FUNCTION_BLOCK FB_PLCopenCall_Test EXTENDS FB_TestSuite
VAR_INPUT
END_VAR
VAR_OUTPUT
END_VAR
VAR
END_VAR

// Copyright (c) 2024 Loupe (https://loupe.team), provided under the MIT License.

Call();
Clear();
Exec();
Start();

METHOD Call
VAR
    call : PLCopenCall;
    command : PLCopenCommand;
END_VAR
// Copyright (c) 2024 Loupe (https://loupe.team), provided under the MIT License.

(*STweep.Disable*)

TEST('PLCopenCallIdle');


	AssertFalse(Condition := call.Busy, Message := 'Busy should be false as default');
	AssertFalse(Condition := call.Done, Message := 'Done should be false as default');
	AssertFalse(Condition := call.Error, Message := 'Error should be false as default');
	
	call.Exec(command);
	AssertTrue(Condition := call.Busy, Message := 'Busy should be true after first exec');
	AssertFalse(Condition := call.Done, Message := 'Done should be false after first exec');
	AssertFalse(Condition := call.Error, Message := 'Error should be false as default');
	AssertEquals_DINT(Expected := PLCopenStatusBase.BUSY, Actual := call.Status, Message := 'Status should be FUB Working');

// new command

// this command aborted

// cleanup

// done

// working

// aborted

// TODO multiple calls
TEST_FINISHED();
END_METHOD

METHOD Clear
VAR
    call : PLCopenCall();
    status : PLCopenStatusBase;
END_VAR
// Copyright (c) 2024 Loupe (https://loupe.team), provided under the MIT License.

(*STweep.Disable*)

TEST('Clear');
	call.Execute := TRUE;
	call();
	status := call.Clear();
	AssertFalse(call.Execute, Message := 'Execute should not be true');
	AssertEquals_INT(Expected := PLCopenStatusBase.NOT_ENABLED, Actual := status, Message := 'Call status should be not enabled');
TEST_FINISHED();
END_METHOD

METHOD Errored
VAR_INPUT
END_VAR
// Copyright (c) 2024 Loupe (https://loupe.team), provided under the MIT License.

(*STweep.Disable*)
END_METHOD

METHOD Exec
VAR
    call : PLCopenCall();
    command1 : PLCopenCommand();
    command2 : PLCopenCommand();
END_VAR
// Copyright (c) 2024 Loupe (https://loupe.team), provided under the MIT License.

(*STweep.Disable*)

TEST('Exec');
	call.Exec(command1);
	AssertTrue(call.Execute, Message := 'Execute should be true');
	
	call.Exec(command2);
	AssertTrue(call.Execute, Message := 'Execute should still be true, second command should abort first');
	AssertFalse(command1.Execute, Message := 'Execute should not be true on first command');
TEST_FINISHED();
END_METHOD

METHOD Start
VAR
    call : PLCopenCall();
    command1 : PLCopenCommand();
    command2 : PLCopenCommand();
END_VAR
// Copyright (c) 2024 Loupe (https://loupe.team), provided under the MIT License.

(*STweep.Disable*)

TEST('Start');
    // TODO check cancelling previous command
	
	// NOTE: since Start is just a wrapper around Exec, these tests are the same as Exec
	call.Start(command1);
	AssertTrue(call.Execute, Message := 'Execute should be true');
	
	call.Start(command2);
	AssertTrue(command1.Execute, Message := 'Execute should not be true on first command');

TEST_FINISHED();
END_METHOD

END_FUNCTION_BLOCK

(* stored: Version 1.1.0.1
   POU FB_PLCopenCall_Test: Id {11b00080-9eb7-435e-b91b-311812c3e08c}, SpecialFunc None
   Method Call: Id {191016cf-95da-4fad-aea1-2f6fad08115d}
   Method Clear: Id {2f219140-8639-4442-9636-f58c99c41e5b}
   Method Errored: Id {a53681cb-16c1-46fc-8764-7d1e04f77a4b}
   Method Exec: Id {ee4d2b03-8c4b-4975-8443-00a2021a958d}
   Method Start: Id {33b29bc8-44e1-4a1e-b951-c14b8679d46f} *)
